{attribute 'qualified_only'}
{attribute 'strict'}
TYPE E_CTRL_MODE_1 :
(
    enum_member := 0
);
END_TYPE

(* stored: Version 1.1.0.1, ProductVersion 3.1.4024.12
   DUT E_CTRL_MODE_1: Id {da0e39c6-ad3a-40af-8e83-e90f801e6208} *)
